// TIA Portal V19 export
FUNCTION "FC_FW_Auftrag_Parken" : Void   // FC186, LAD
{ S7_Optimized_Access := 'TRUE' }
// stored: AutoNumber false, SetENOAutomatically false
   VAR_OUTPUT
      nextStep : Bool;
      startStep : Bool;
   END_VAR
   VAR_IN_OUT
      Quelle : Int;
      Ziel : Int;
      Positionen : Array[1..30] of "UDT_Auftrag_Pos";
   END_VAR
   VAR_TEMP
      Befehl_ok : Bool;
   END_VAR
BEGIN

REGION Network 1 (SCL)
   IF (#Quelle <> 0) AND (#Ziel <> 0) THEN
       #nextStep := #Positionen[#Quelle].Sperre;
       #startStep := NOT #nextStep;
       #Quelle := 0;
       #Ziel := 0;
       RETURN;
   END_IF;

   #Quelle := 0;
   #Ziel := 0;
   #nextStep := FALSE;
   #startStep := FALSE;
END_REGION

REGION Network 2 (SCL): Transportwagen schieben
   //CM01
   IF ("DI_FW_1".ZST.POSITION_li <= 6) THEN
       "FC_FW_Auftrag_Befehl"(inQuelle := 7,
                              inZiel := 0,
                              Befehl_ok => #Befehl_ok,
                              outQuelle => #Quelle,
                              outZiel => #Ziel);

       #nextStep := NOT #Befehl_ok;
       RETURN;
   END_IF;

   //CM02
   IF ("DI_FW_1".ZST.POSITION_li >= 13) AND ("DI_FW_1".ZST.POSITION_li <= 18) THEN
       "FC_FW_Auftrag_Befehl"(inQuelle := 11,
                              inZiel := 0,
                              Befehl_ok => #Befehl_ok,
                              outQuelle => #Quelle,
                              outZiel => #Ziel);

       #nextStep := NOT #Befehl_ok;
       RETURN;
   END_IF;

   //WR02
   IF ("DI_FW_1".ZST.POSITION_li >= 25) THEN
       "FC_FW_Auftrag_Befehl"(inQuelle := 23,
                              inZiel := 0,
                              Befehl_ok => #Befehl_ok,
                              outQuelle => #Quelle,
                              outZiel => #Ziel);

       #nextStep := NOT #Befehl_ok;
       RETURN;
   END_IF;

   //?
   #nextStep := TRUE;
END_REGION
END_FUNCTION
